% RSLogix 500 project P9.RSS, saved by version 8.30.00.16 %
PROJECT "UNTITLED"    % processor: Bul.1763 MicroLogix 1100 Series B %

PROGRAM FILES
  LAD 2   8 rungs

DATA FILES
  O0 OUTPUT  4 elements
  I1 INPUT  6 elements
  S2 STATUS  66 elements
  B3 BINARY  1 elements
  T4 TIMER  1 elements
  C5 COUNTER  1 elements
  R6 CONTROL  1 elements
  N7 INTEGER  4 elements
  F8 FLOAT  1 elements
  ST9 STRING  8 elements

LADDER 2
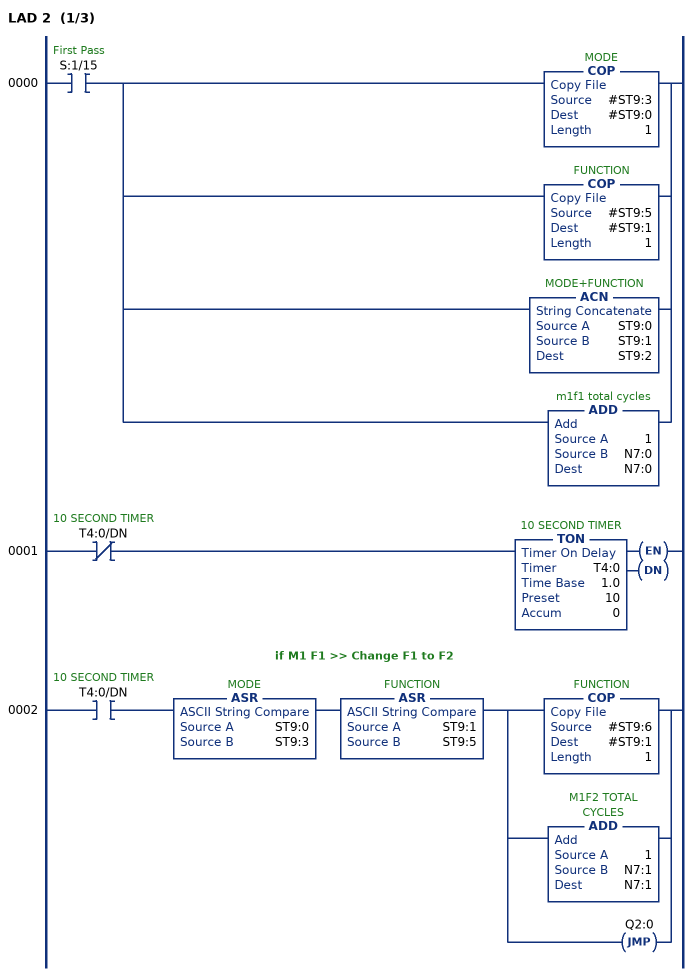
% Rung: 0 %
SOR XIC S:1/15 BST COP #ST9:3 #ST9:0 1 NXB COP #ST9:5 #ST9:1 1 NXB ACN ST9:0 ST9:1 ST9:2 NXB ADD 1 N7:0 N7:0 BND EOR
%   S:1/15  "First Pass" %
%   ST9:3  "Start with Mode 1" %
%   ST9:0  "MODE" %
%   ST9:5  "F1" %
%   ST9:1  "FUNCTION" %
%   ST9:2  "MODE+FUNCTION" %
%   N7:0  "m1f1 total cycles" %
% Rung: 1 %
SOR XIO T4:0/DN TON T4:0 1.0 10 0 EOR
%   T4:0  "10 SECOND TIMER" %
% Rung: 2 %
% TITLE: if M1 F1 >> Change F1 to F2 %
SOR XIC T4:0/DN ASR ST9:0 ST9:3 ASR ST9:1 ST9:5 BST COP #ST9:6 #ST9:1 1 NXB ADD 1 N7:1 N7:1 NXB JMP Q2:0 BND EOR
%   T4:0  "10 SECOND TIMER" %
%   ST9:0  "MODE" %
%   ST9:3  "Start with Mode 1" %
%   ST9:1  "FUNCTION" %
%   ST9:5  "F1" %
%   ST9:6  "F2" %
%   N7:1  "M1F2 TOTAL CYCLES" %

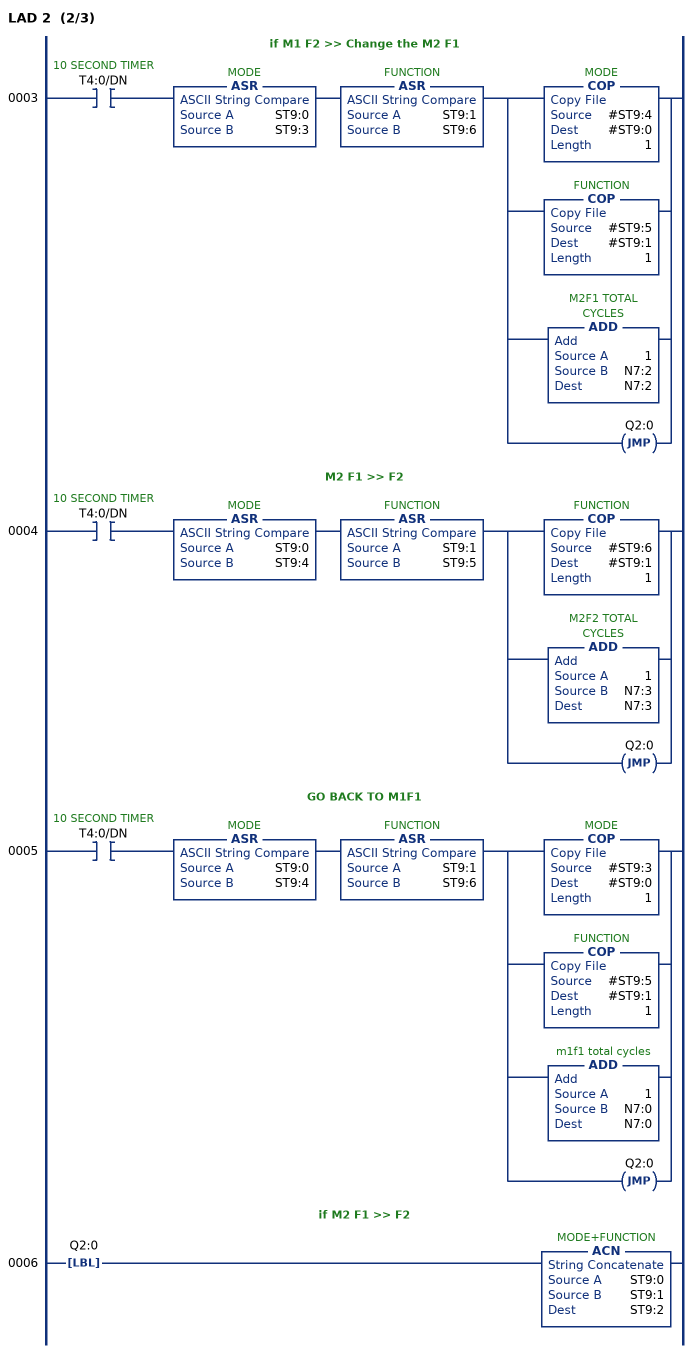
% Rung: 3 %
% TITLE: if M1 F2 >> Change the M2 F1 %
SOR XIC T4:0/DN ASR ST9:0 ST9:3 ASR ST9:1 ST9:6 BST COP #ST9:4 #ST9:0 1 NXB COP #ST9:5 #ST9:1 1 NXB ADD 1 N7:2 N7:2 NXB JMP Q2:0 BND EOR
%   T4:0  "10 SECOND TIMER" %
%   ST9:0  "MODE" %
%   ST9:3  "Start with Mode 1" %
%   ST9:1  "FUNCTION" %
%   ST9:6  "F2" %
%   ST9:5  "F1" %
%   N7:2  "M2F1 TOTAL CYCLES" %
% Rung: 4 %
% TITLE: M2 F1 >> F2 %
SOR XIC T4:0/DN ASR ST9:0 ST9:4 ASR ST9:1 ST9:5 BST COP #ST9:6 #ST9:1 1 NXB ADD 1 N7:3 N7:3 NXB JMP Q2:0 BND EOR
%   T4:0  "10 SECOND TIMER" %
%   ST9:0  "MODE" %
%   ST9:1  "FUNCTION" %
%   ST9:5  "F1" %
%   ST9:6  "F2" %
%   N7:3  "M2F2 TOTAL CYCLES" %
% Rung: 5 %
% TITLE: GO BACK TO M1F1 %
SOR XIC T4:0/DN ASR ST9:0 ST9:4 ASR ST9:1 ST9:6 BST COP #ST9:3 #ST9:0 1 NXB COP #ST9:5 #ST9:1 1 NXB ADD 1 N7:0 N7:0 NXB JMP Q2:0 BND EOR
%   T4:0  "10 SECOND TIMER" %
%   ST9:0  "MODE" %
%   ST9:1  "FUNCTION" %
%   ST9:6  "F2" %
%   ST9:3  "Start with Mode 1" %
%   ST9:5  "F1" %
%   N7:0  "m1f1 total cycles" %
% Rung: 6 %
% TITLE: if M2 F1 >> F2 %
SOR LBL Q2:0 ACN ST9:0 ST9:1 ST9:2 EOR
%   ST9:0  "MODE" %
%   ST9:1  "FUNCTION" %
%   ST9:2  "MODE+FUNCTION" %

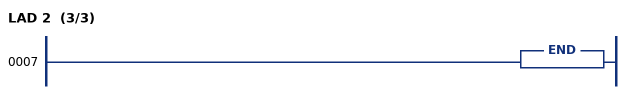
% Rung: 7 %
SOR END EOR

OTHER DOCUMENTED ADDRESSES
  B3:0/0  "place holder"

DATA TABLE (non-zero values as saved)
DATA T4
% .PRE .ACC %
% T4:0 % 10 0
DATA ST9
% ST9:3 % "Mode-1 "
% ST9:4 % "Mode-2 "
% ST9:5 % "F1"
% ST9:6 % "F2"
